// Mitsubishi GX Works2 project: EX2_PLC_Final   PLC: FX3G

// global labels: Global1
VAR_GLOBAL
  Start_Workday_Switch AT X007 : BOOL;
  Workday_Lamp AT Y007 : BOOL;
  Emergency_Stop AT X005 : BOOL;
  Cooling_Switch AT X002 : BOOL;
  Start_Prep_Switch AT X001 : BOOL;
  Temp_Sensor AT X003 : BOOL;
  Prep_Lamp AT Y000 : BOOL;
  Cooling_Lamp AT Y002 : BOOL;
  Mixing_Lamp_A AT Y005 : BOOL;
  Mixing_Lamp_B AT Y006 : BOOL;
  M_Workday_On AT M0 : BOOL;
  M_Is_Treat_Pack AT M1 : BOOL;
  M_Low_Stock_Error AT M2 : BOOL;
  Stock_Raspberry AT D1100 : REAL;
  Stock_Lemon AT D1110 : REAL;
  Stock_Stabilizer AT D1120 : REAL;
  Stock_Gummy_Bears AT D1130 : REAL;
  Storage_Inventory AT D1150 : REAL;
  Timer_Prep AT TC0 : BOOL;
  Timer_Cooling AT TC1 : BOOL;
  Timer_Mixing_Treat AT TC2 : BOOL;
  Timer_Flash_1 AT TC3 : BOOL;
  Timer_Flash_2 AT TC4 : BOOL;
END_VAR
VAR_GLOBAL CONSTANT
  K_Prep_Time : INT := 50;
  K_Max_Cool_Time : INT := 80;
  K_Mix_Reg_Time : INT := 30;
  K_Mix_Treat_Time : INT := 50;
  K_Flash_Interval : INT := 5;
END_VAR
VAR_GLOBAL
  Analog_In_Selector AT D8280 : INT;
  Analog_Out_Total AT D8282 : INT;
  M_Mixing_Phase AT M3 : BOOL;
  M_Flash_Enable AT M4 : BOOL;
  Init_Stock_Raspberry AT D1000 : REAL;
  Init_Stock_Lemon AT D1010 : REAL;
  Init_Stock_Stabilizer AT D1020 : REAL;
  Init_Stock_Gummy_Bears AT D1030 : REAL;
  Sampled_Analog_Val AT D1170 : REAL;
  Prep_Tank_Raspberry AT D1040 : REAL;
  Prep_Tank_Lemon AT D1050 : REAL;
  Cool_Tank_Raspberry AT D1060 : REAL;
  Cool_Tank_Lemon AT D1070 : REAL;
  M_Cool_Raspberry AT M5 : BOOL;
  M_Cool_Lemon AT M6 : BOOL;
  Mix_Tank AT D1080 : REAL;
  Pack_Counter_Float AT D1140 : REAL;
  Converted_Result AT D1180 : REAL;
  M_Workday_Off AT M10 : BOOL;
  Is_Treat_Lamp AT Y001 : BOOL;
  Operation_Error_Lamp AT Y004 : BOOL;
  M_Prep_Done AT M7 : BOOL;
  M_Operation_Eror AT M8 : BOOL;
  Timer_Mixing_Reg AT TC5 : BOOL;
  M_Finish_Mixing_Phase AT M9 : BOOL;
  Stop_Operation_Error AT M11 : BOOL;
END_VAR

// task Task_01 (event TRUE, interval 0, priority 31): POU_01

PROGRAM POU_01
VAR
  TC2 : BOOL;
END_VAR
(* structured ladder/FBD written out as ST: instructions are called as NAME(EN, inputs, outputs); _pN, _eN, _tN stand for wires *)
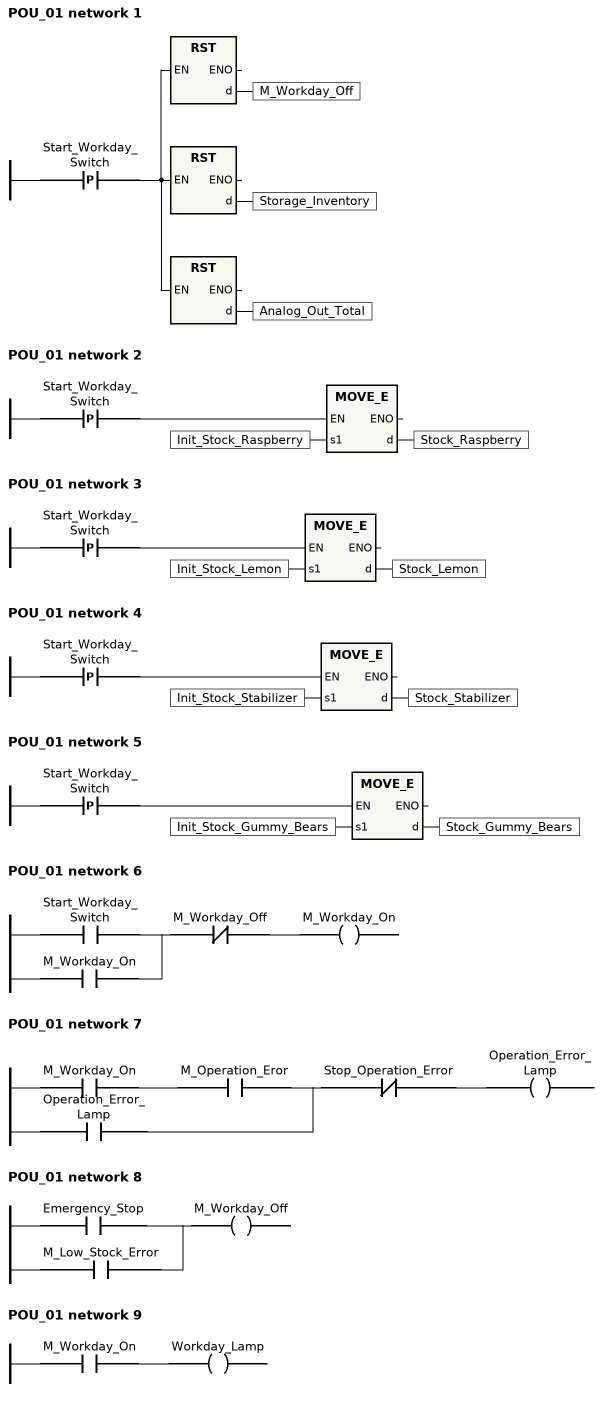
(* network 1 *)
_p1 := LDP(TRUE, Start_Workday_Switch);
RST(_p1, M_Workday_Off);
RST(_p1, Storage_Inventory);
RST(_p1, Analog_Out_Total);
(* network 2 *)
MOVE_E(LDP(TRUE, Start_Workday_Switch), Init_Stock_Raspberry, Stock_Raspberry);
(* network 3 *)
MOVE_E(LDP(TRUE, Start_Workday_Switch), Init_Stock_Lemon, Stock_Lemon);
(* network 4 *)
MOVE_E(LDP(TRUE, Start_Workday_Switch), Init_Stock_Stabilizer, Stock_Stabilizer);
(* network 5 *)
MOVE_E(LDP(TRUE, Start_Workday_Switch), Init_Stock_Gummy_Bears, Stock_Gummy_Bears);
(* network 6 *)
M_Workday_On := (Start_Workday_Switch OR M_Workday_On) AND NOT M_Workday_Off;
(* network 7 *)
Operation_Error_Lamp := ((M_Workday_On AND M_Operation_Eror) OR Operation_Error_Lamp) AND NOT Stop_Operation_Error;
(* network 8 *)
M_Workday_Off := Emergency_Stop OR M_Low_Stock_Error;
(* network 9 *)
Workday_Lamp := M_Workday_On;
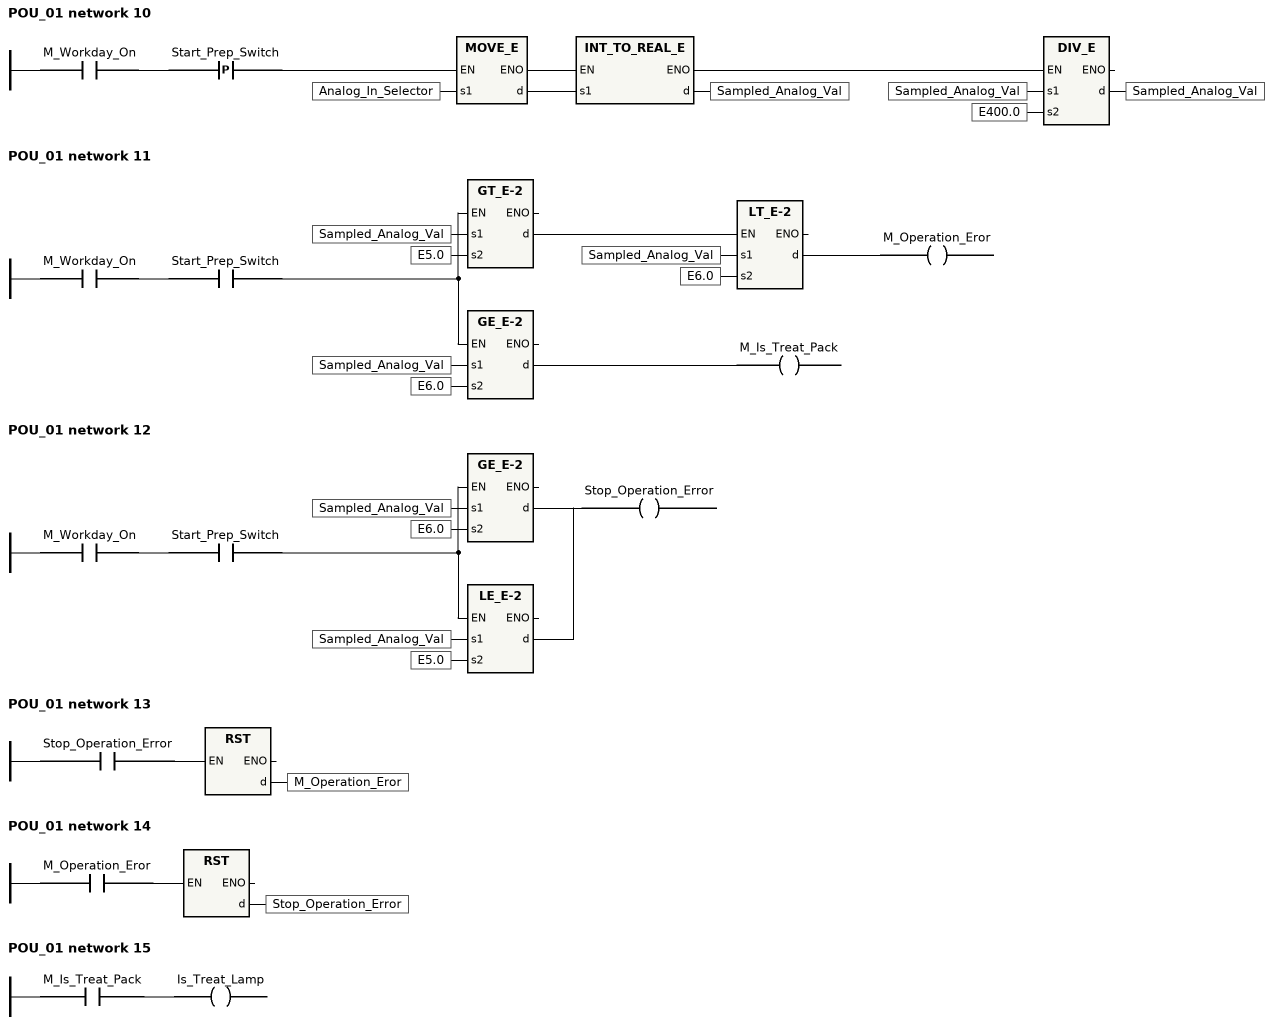
(* network 10 *)
_e2 := MOVE_E(M_Workday_On AND LDP(TRUE, Start_Prep_Switch), Analog_In_Selector, _t1);
_e3 := INT_TO_REAL_E(_e2, _t1, Sampled_Analog_Val);
DIV_E(_e3, Sampled_Analog_Val, E400.0, Sampled_Analog_Val);
(* network 11 *)
_p1 := M_Workday_On AND Start_Prep_Switch;
GE_E(_p1, Sampled_Analog_Val, E6.0, _t2);
M_Is_Treat_Pack := _t2;
GT_E(_p1, Sampled_Analog_Val, E5.0, _t3);
LT_E(_t3, Sampled_Analog_Val, E6.0, _t4);
M_Operation_Eror := _t4;
(* network 12 *)
_p1 := M_Workday_On AND Start_Prep_Switch;
GE_E(_p1, Sampled_Analog_Val, E6.0, _t2);
LE_E(_p1, Sampled_Analog_Val, E5.0, _t3);
Stop_Operation_Error := _t2 OR _t3;
(* network 13 *)
RST(Stop_Operation_Error, M_Operation_Eror);
(* network 14 *)
RST(M_Operation_Eror, Stop_Operation_Error);
(* network 15 *)
Is_Treat_Lamp := M_Is_Treat_Pack;
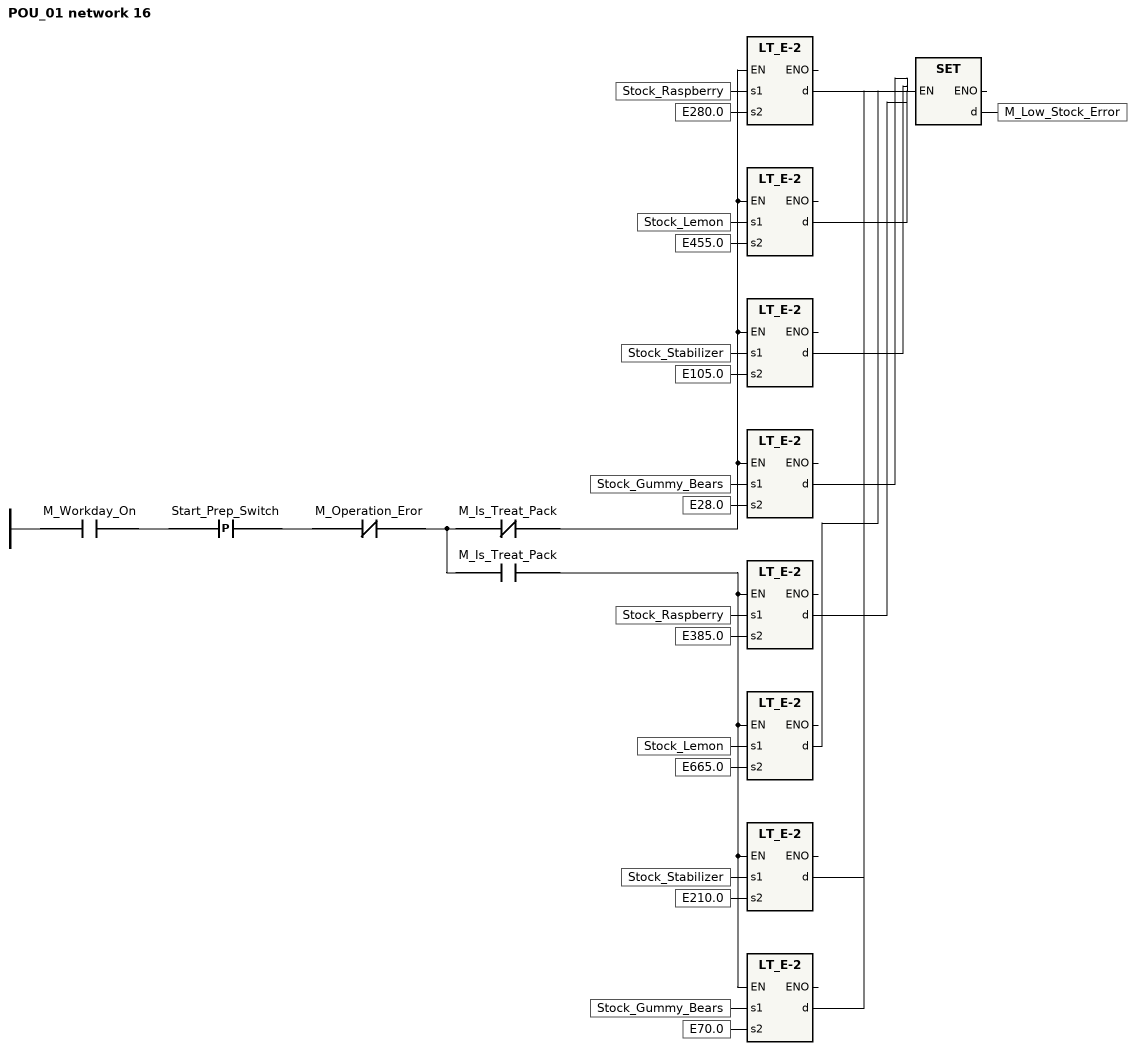
(* network 16 *)
_p1 := M_Workday_On AND LDP(TRUE, Start_Prep_Switch) AND NOT M_Operation_Eror;
_p2 := _p1 AND NOT M_Is_Treat_Pack;
LT_E(_p2, Stock_Raspberry, E280.0, _t3);
LT_E(_p2, Stock_Lemon, E455.0, _t4);
LT_E(_p2, Stock_Stabilizer, E105.0, _t5);
LT_E(_p2, Stock_Gummy_Bears, E28.0, _t6);
_p7 := _p1 AND M_Is_Treat_Pack;
LT_E(_p7, Stock_Raspberry, E385.0, _t8);
LT_E(_p7, Stock_Lemon, E665.0, _t9);
LT_E(_p7, Stock_Stabilizer, E210.0, _t10);
LT_E(_p7, Stock_Gummy_Bears, E70.0, _t11);
SET(_t3 OR _t4 OR _t5 OR _t6 OR _t8 OR _t9 OR _t10 OR _t11, M_Low_Stock_Error);
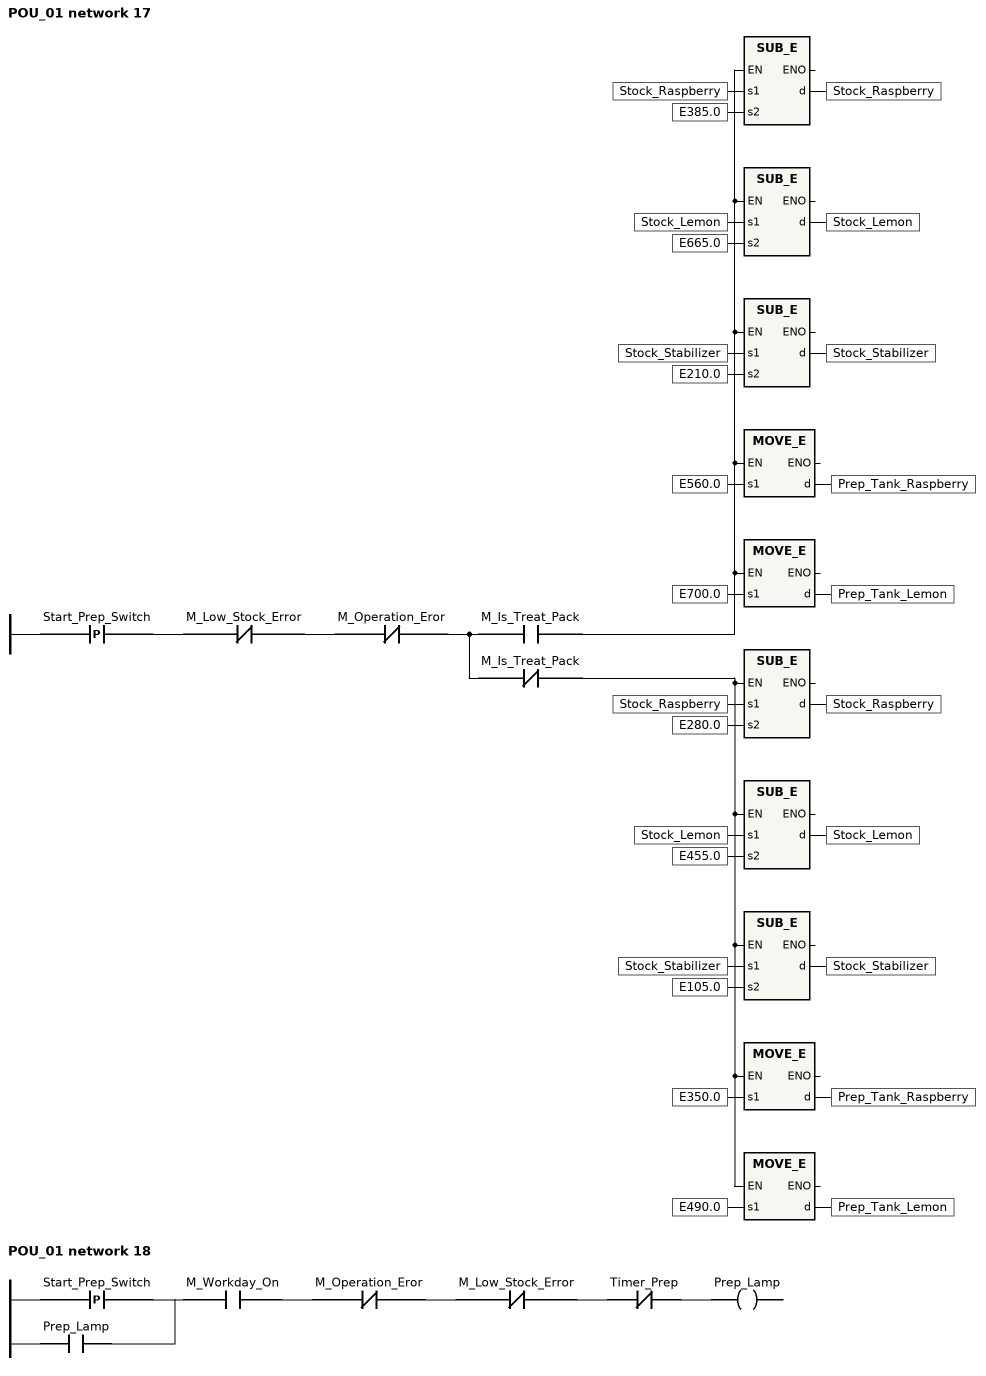
(* network 17 *)
_p1 := LDP(TRUE, Start_Prep_Switch) AND NOT M_Low_Stock_Error AND NOT M_Operation_Eror;
_p2 := _p1 AND M_Is_Treat_Pack;
SUB_E(_p2, Stock_Raspberry, E385.0, Stock_Raspberry);
SUB_E(_p2, Stock_Lemon, E665.0, Stock_Lemon);
SUB_E(_p2, Stock_Stabilizer, E210.0, Stock_Stabilizer);
MOVE_E(_p2, E560.0, Prep_Tank_Raspberry);
MOVE_E(_p2, E700.0, Prep_Tank_Lemon);
_p3 := _p1 AND NOT M_Is_Treat_Pack;
SUB_E(_p3, Stock_Raspberry, E280.0, Stock_Raspberry);
SUB_E(_p3, Stock_Lemon, E455.0, Stock_Lemon);
SUB_E(_p3, Stock_Stabilizer, E105.0, Stock_Stabilizer);
MOVE_E(_p3, E350.0, Prep_Tank_Raspberry);
MOVE_E(_p3, E490.0, Prep_Tank_Lemon);
(* network 18 *)
Prep_Lamp := ((((LDP(TRUE, Start_Prep_Switch) OR Prep_Lamp) AND M_Workday_On) AND NOT M_Operation_Eror) AND NOT M_Low_Stock_Error) AND NOT Timer_Prep;
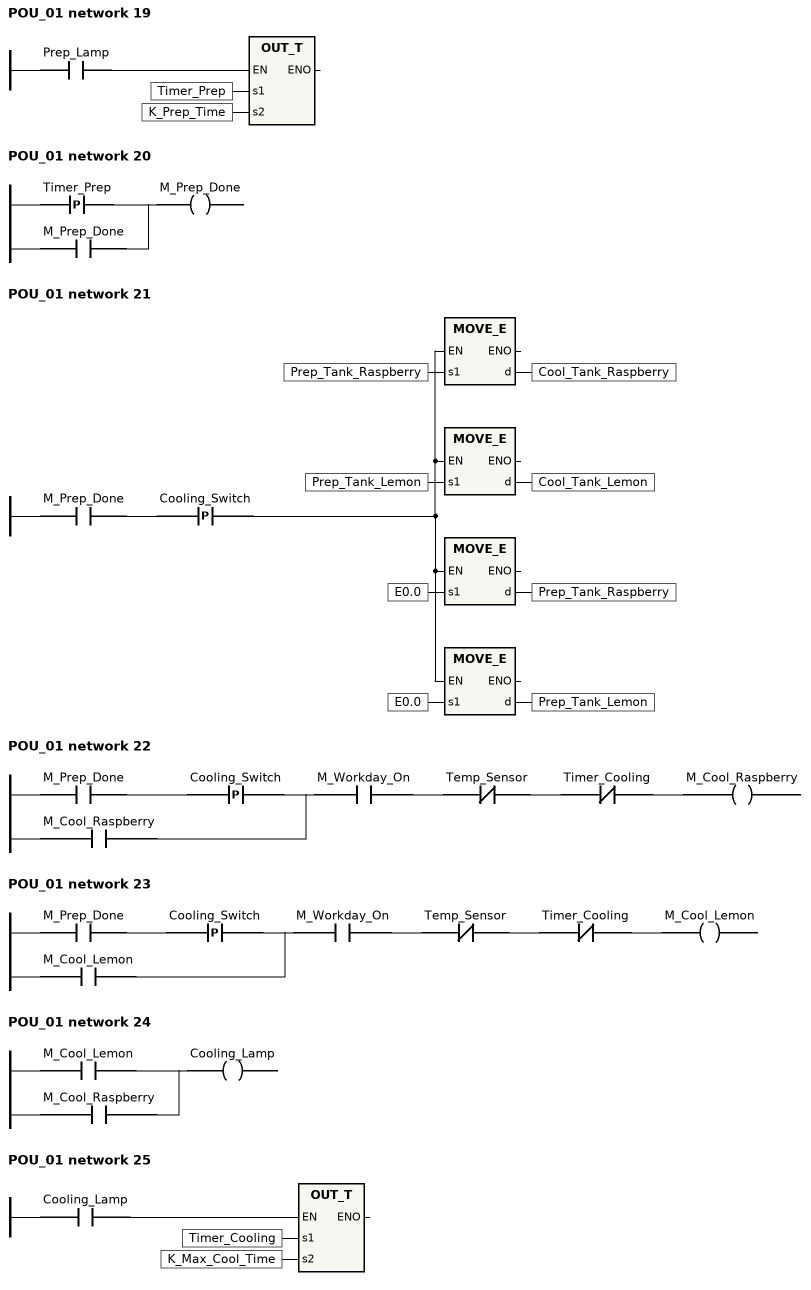
(* network 19 *)
OUT_T(Prep_Lamp, Timer_Prep, K_Prep_Time);
(* network 20 *)
M_Prep_Done := LDP(TRUE, Timer_Prep) OR M_Prep_Done;
(* network 21 *)
_p1 := M_Prep_Done AND LDP(TRUE, Cooling_Switch);
MOVE_E(_p1, Prep_Tank_Raspberry, Cool_Tank_Raspberry);
MOVE_E(_p1, Prep_Tank_Lemon, Cool_Tank_Lemon);
MOVE_E(_p1, E0.0, Prep_Tank_Raspberry);
MOVE_E(_p1, E0.0, Prep_Tank_Lemon);
(* network 22 *)
M_Cool_Raspberry := ((((M_Prep_Done AND LDP(TRUE, Cooling_Switch)) OR M_Cool_Raspberry) AND M_Workday_On) AND NOT Temp_Sensor) AND NOT Timer_Cooling;
(* network 23 *)
M_Cool_Lemon := ((((M_Prep_Done AND LDP(TRUE, Cooling_Switch)) OR M_Cool_Lemon) AND M_Workday_On) AND NOT Temp_Sensor) AND NOT Timer_Cooling;
(* network 24 *)
Cooling_Lamp := M_Cool_Lemon OR M_Cool_Raspberry;
(* network 25 *)
OUT_T(Cooling_Lamp, Timer_Cooling, K_Max_Cool_Time);
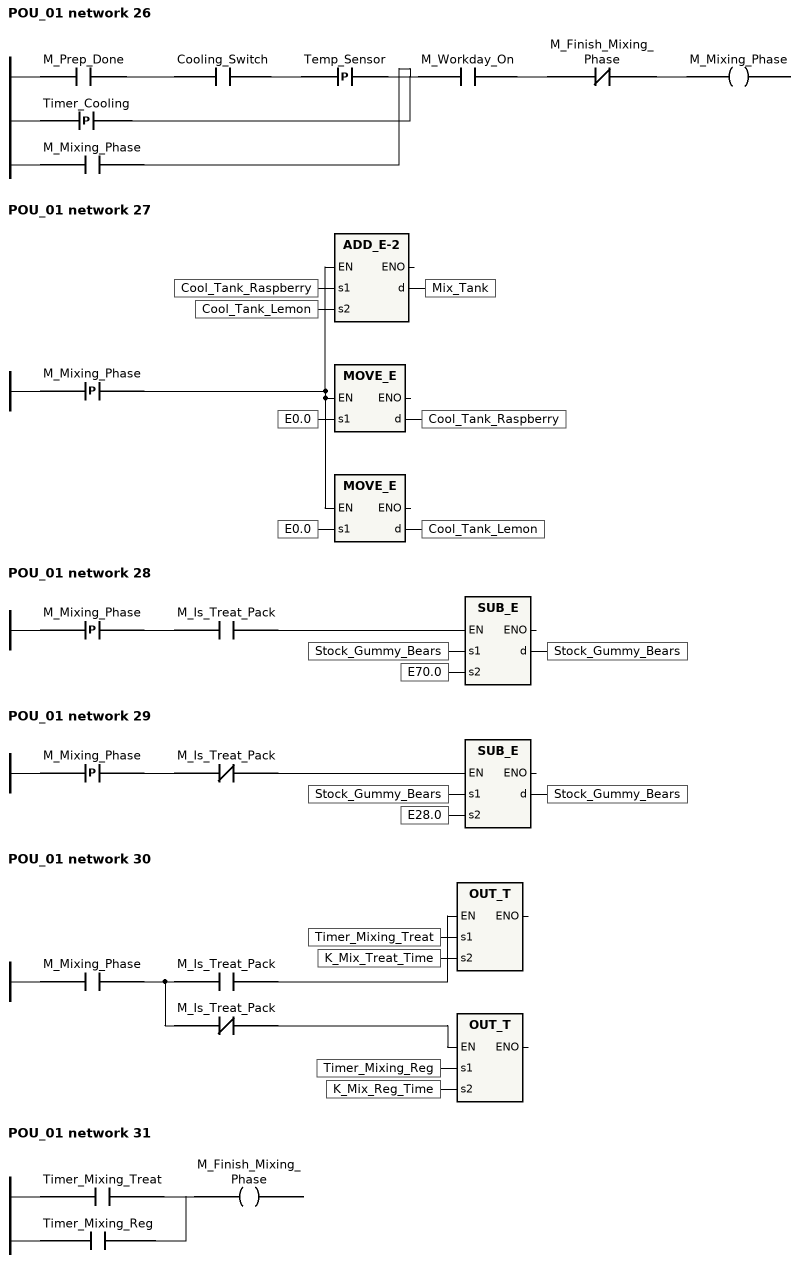
(* network 26 *)
M_Mixing_Phase := (((M_Prep_Done AND Cooling_Switch AND LDP(TRUE, Temp_Sensor)) OR LDP(TRUE, Timer_Cooling) OR M_Mixing_Phase) AND M_Workday_On) AND NOT M_Finish_Mixing_Phase;
(* network 27 *)
_p1 := LDP(TRUE, M_Mixing_Phase);
ADD_E(_p1, Cool_Tank_Raspberry, Cool_Tank_Lemon, Mix_Tank);
MOVE_E(_p1, E0.0, Cool_Tank_Raspberry);
MOVE_E(_p1, E0.0, Cool_Tank_Lemon);
(* network 28 *)
SUB_E(LDP(TRUE, M_Mixing_Phase) AND M_Is_Treat_Pack, Stock_Gummy_Bears, E70.0, Stock_Gummy_Bears);
(* network 29 *)
SUB_E(LDP(TRUE, M_Mixing_Phase) AND NOT M_Is_Treat_Pack, Stock_Gummy_Bears, E28.0, Stock_Gummy_Bears);
(* network 30 *)
OUT_T(M_Mixing_Phase AND M_Is_Treat_Pack, Timer_Mixing_Treat, K_Mix_Treat_Time);
OUT_T(M_Mixing_Phase AND NOT M_Is_Treat_Pack, Timer_Mixing_Reg, K_Mix_Reg_Time);
(* network 31 *)
M_Finish_Mixing_Phase := Timer_Mixing_Treat OR Timer_Mixing_Reg;
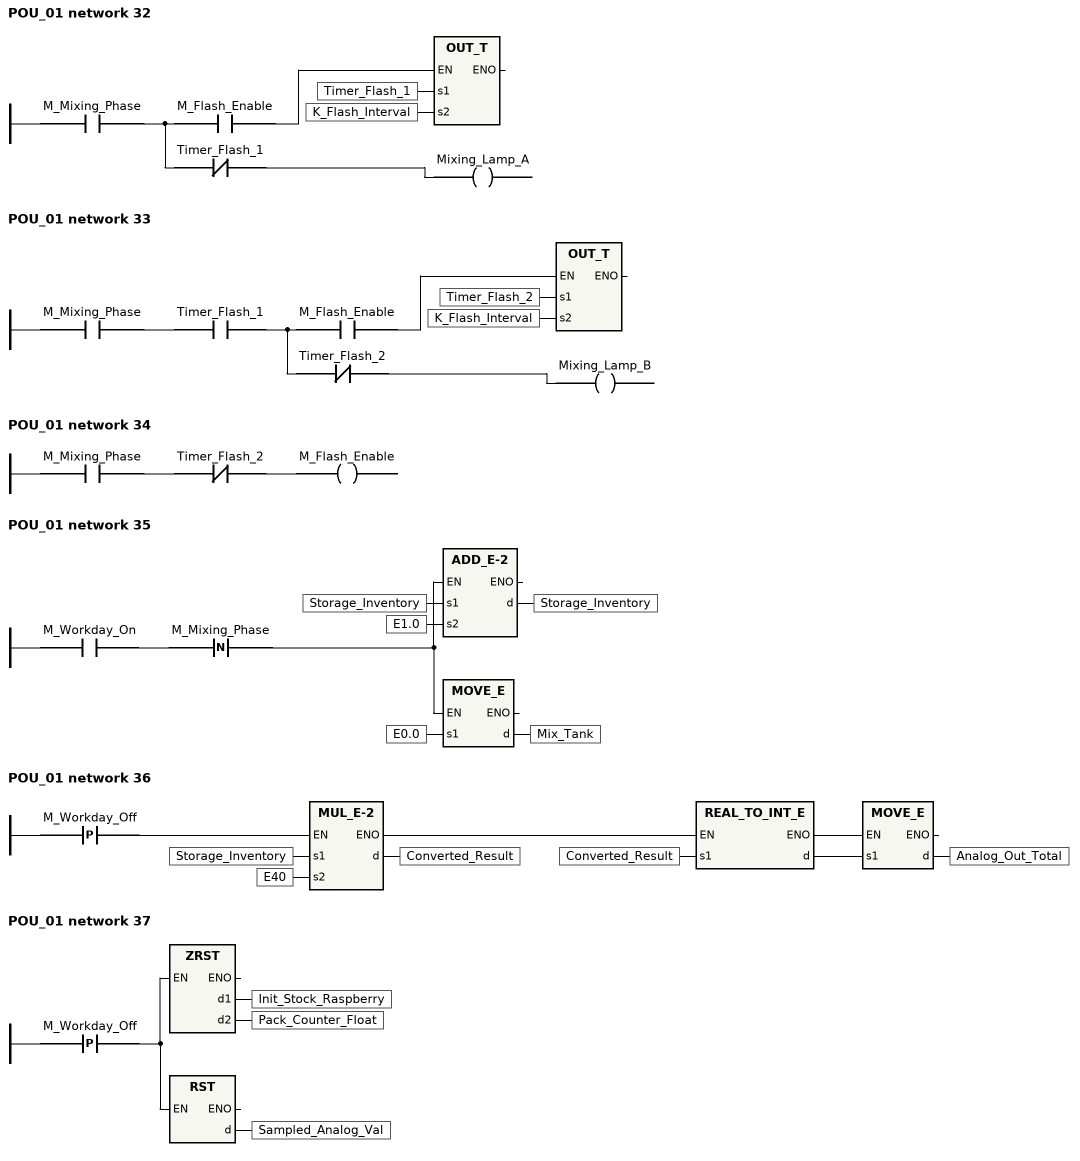
(* network 32 *)
OUT_T(M_Mixing_Phase AND M_Flash_Enable, Timer_Flash_1, K_Flash_Interval);
Mixing_Lamp_A := M_Mixing_Phase AND NOT Timer_Flash_1;
(* network 33 *)
_p1 := M_Mixing_Phase AND Timer_Flash_1;
OUT_T(_p1 AND M_Flash_Enable, Timer_Flash_2, K_Flash_Interval);
Mixing_Lamp_B := _p1 AND NOT Timer_Flash_2;
(* network 34 *)
M_Flash_Enable := M_Mixing_Phase AND NOT Timer_Flash_2;
(* network 35 *)
_p1 := M_Workday_On AND LDF(TRUE, M_Mixing_Phase);
ADD_E(_p1, Storage_Inventory, E1.0, Storage_Inventory);
MOVE_E(_p1, E0.0, Mix_Tank);
(* network 36 *)
_e1 := MUL_E(LDP(TRUE, M_Workday_Off), Storage_Inventory, E40, Converted_Result);
_e3 := REAL_TO_INT_E(_e1, Converted_Result, _t2);
MOVE_E(_e3, _t2, Analog_Out_Total);
(* network 37 *)
_p1 := LDP(TRUE, M_Workday_Off);
ZRST(_p1, Init_Stock_Raspberry, Pack_Counter_Float);
RST(_p1, Sampled_Analog_Val);
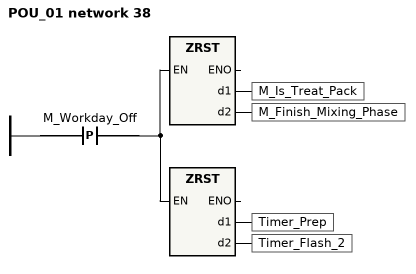
(* network 38 *)
_p1 := LDP(TRUE, M_Workday_Off);
ZRST(_p1, M_Is_Treat_Pack, M_Finish_Mixing_Phase);
ZRST(_p1, Timer_Prep, Timer_Flash_2);
END_PROGRAM
